INTERFACE Message

METHOD Send
VAR_INPUT
END_VAR
END_METHOD

{attribute 'monitoring' := 'call'}
PROPERTY Source : Name
GET
END_GET
SET
END_SET
END_PROPERTY

END_INTERFACE

(* stored: Version 1.1.0.1, ProductVersion 3.1.4024.15
   Itf Message: Id {43a9cf12-ef21-0d83-2603-50b2d81d5535}
   Method Send: Id {a97dd082-ac5b-03e1-2dae-4e3bad4af412}
   Property Source: Id {d1c99de6-7f60-06fe-27bf-07c114b4cffe}
   Get Get: Id {4b178a5b-1417-088e-3a8c-66902242b841}
   Set Set: Id {b7feb3fa-4042-0a08-33d7-0d7838edc479} *)
